TYPE ST_DigitalInputIO :
STRUCT
	stIn 	AT%I* : ST_DigitalInputIn;
END_STRUCT
END_TYPE

(* stored: Version 1.1.0.1, ProductVersion 3.1.4022.9
   DUT ST_DigitalInputIO: Id {7a132cb5-0a79-49e4-ac0e-f3f2e780e2b3} *)
